PROGRAM P_PID
VAR
	fbPID : FB_PID;
	fbIntegrator : FB_Integrator;
	fbDerivator : FB_Derivator;
	fbDerivatorFiltering : FB_Filtering;
END_VAR


fbPID(
	fX := G_OPC.fXRef,
	fXReal := G_OPC.fPistonPosition,
		
	fError => G_OPC.fError
);

IF (G_Enables.bEnablePID AND G_Mode.bRunning) THEN
	
	fbDerivatorFiltering(
		ssMethodType := 1,
		Signal := fbPID.fSignalD,
		Num := G_FilterConstants.fDerivatorFilterNum,
		Denz := G_FilterConstants.fDerivatorFilterDenz,
		Den := G_FilterConstants.fDerivatorFilterDen,
		Initial := G_FilterConstants.fDerivatorFilterInit,
		Signal_Filtered => fbDerivator.fSignal
	);
	
	fbIntegrator(
		ssMethodType := BOOL_TO_SINT(G_Inputs.bStartButton),
		fSignal := fbPID.fSignalI,
		fSignalIntegrated => fbPID.fSignalIntegrated
	);
	fbDerivator(
		ssMethodType := BOOL_TO_SINT(G_Inputs.bStartButton),
		fSignal := fbPID.fSignalD,
		fSignalDerivative => fbPID.fSignalDerivated
	);

	fbPID(
		bEnablePID := G_Enables.bEnablePID,
		fX := G_OPC.fXRef,
		fXReal := G_OPC.fPistonPosition,
		fKp := G_Parameter.Kp,
		fKi := G_Parameter.Ki,
		fKd := G_Parameter.Kd,
		
		fSignalAdjusted => G_OPC.fSignalPID
	);

END_IF

END_PROGRAM

(* stored: Version 1.1.0.1, ProductVersion 3.1.4024.12
   POU P_PID: Id {8618f120-26c6-4eb7-b274-74ff26057632}, SpecialFunc None *)
